{attribute 'qualified_only'}
VAR_GLOBAL
	DO1_1 : BOOL; 
END_VAR

(* stored: Version 1.1.0.1, ProductVersion 3.1.4024.9
   GVL Outputs: Id {8632dc2c-f2e8-400e-b1a8-ffb8dbbb7ffb} *)
